SUBAPPLICATION ResetDemo (* Reset pattern demo: RESET drives its own TrueUntil directly, bypassing the E_SR/E_PERMIT start/stop gate that guards the normal TRIGGER path *)
  (* Standard: 61499-2; Description: Copyright (c) 2026 Meisterschulen am Ostbahnhof This program and the accompanying materials are made available under the terms of the Eclipse Public License 2.0 which is available at https://www.eclipse.org/legal/epl-2.0/ SPDX-License-Identifier: EPL-2.0 *)
  (* Version 1.0, 2026-08-31, Franz Höpfinger, Meisterschulen am Ostbahnhof, Reset design pattern (IEC 61499 primer course, Module 6, Valeriy Vyatkin, slide 71), demo application *)
  PACKAGE Meins::DesingPatterns::ResetPattern;
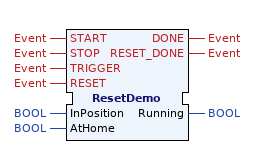
  EVENT_INPUT
    START; (* Start the plant: opens the permit gate for the normal TRIGGER path *)
    STOP; (* Stop the plant: closes the permit gate for the normal TRIGGER path *)
    TRIGGER; (* Ask the normal step to run - only reaches it while the plant is started *)
    RESET; (* Ask the reset step to run - bypasses the start/stop gate entirely, works even while stopped *)
  END_EVENT
  EVENT_OUTPUT
    DONE; (* The normal step completed *)
    RESET_DONE; (* The reset step completed *)
  END_EVENT
  VAR_INPUT
    InPosition : BOOL; (* Demo: simulate the normal step's actuator reaching its position *)
    AtHome : BOOL; (* Demo: simulate the reset step's actuator reaching the home position *)
  END_VAR
  VAR_OUTPUT
    Running : BOOL; (* Current start/stop state (E_SR.Q): TRUE while the plant is started - RESET ignores this *)
  END_VAR
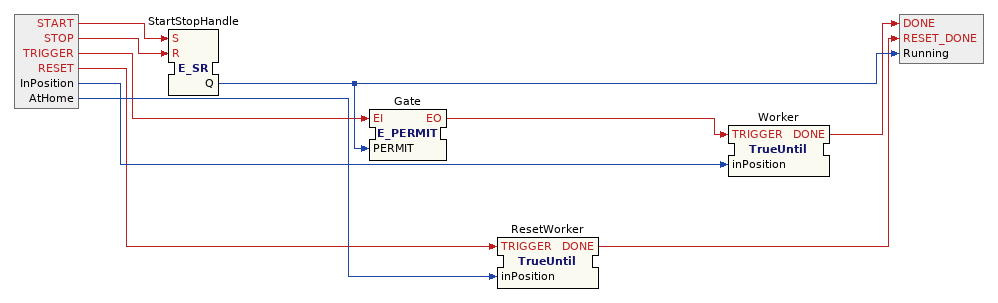
  FBS
    StartStopHandle : iec61499::events::E_SR;
    Gate : iec61499::events::E_PERMIT;
    Worker : Meins::DesingPatterns::ChainOfActionsPattern::TrueUntil;
    ResetWorker : Meins::DesingPatterns::ChainOfActionsPattern::TrueUntil;
  END_FBS
  EVENT_CONNECTIONS
    START TO StartStopHandle.S;
    STOP TO StartStopHandle.R;
    TRIGGER TO Gate.EI;
    Gate.EO TO Worker.TRIGGER;
    Worker.DONE TO DONE;
    RESET TO ResetWorker.TRIGGER; (* Bypasses StartStopHandle/Gate entirely - works even while stopped *)
    ResetWorker.DONE TO RESET_DONE;
  END_CONNECTIONS
  DATA_CONNECTIONS
    StartStopHandle.Q TO Gate.PERMIT;
    StartStopHandle.Q TO Running;
    InPosition TO Worker.inPosition;
    AtHome TO ResetWorker.inPosition;
  END_CONNECTIONS
END_SUBAPPLICATION
